// TIA Portal V20 export
// export: Created 2025-12-01T14:56:19.1590211Z, ExportSetting None, DisplayName Totally Integrated Automation Portal, DisplayVersion V20 Update 3, DisplayName TIA Portal Openness, DisplayVersion V20 Update 3, DisplayName TIA Portal Version Control Interface, DisplayVersion V20 Update 3, DisplayName STEP 7 Professional, DisplayVersion V20 Update 3, DisplayName STEP 7 Safety, DisplayVersion V20 Update 2, DisplayName WinCC Basic/Comfort/Advanced, DisplayVersion V20 Update 3, DisplayName WinCC Professional, DisplayVersion V20 Update 3, DisplayName WinCC Unified, DisplayVersion V20 Update 3
TYPE "i550 Palabra de control"
   STRUCT
      "Reserva 1" : Bool;
      "Reserva 2" : Bool;
      "Reserva 3" : Bool;
      "Reserva 4" : Bool;
      "Reserva 5" : Bool;
      "Reserva 6" : Bool;
      "Reserva 7" : Bool;
      "Reserva 8" : Bool;
      "Run forward" : Bool;   // Avanzar
      "Reverse rotation dirtect." : Bool;   // Avanzar en sentido inverso (junto con Run forward)
      "Reset error" : Bool;   // Resetear fallo en variador
      "Position counter reset" : Bool;   // Resetear valor de cota (solo con encoder)
      "Activate quick stop" : Bool;   // Activar parada rápida controlada
      "Sel. paramset b0" : Bool;   // Variable 0 para cambio de parámetros
      "Sel. paramset b1" : Bool;   // Variable 1 para cambio de parámetros
      "Activar salida DO1" : Bool;   // Activa la salida DO1 (solo en caso de no tener freno equipado)
   END_STRUCT;
END_TYPE
